PROGRAM SDOMotorErrorFlags
VAR
	ErrorFlagsKlemme1: getSDOMotorErrorFlags;
	ErrorFlagsKlemme2: getSDOMotorErrorFlags;
END_VAR

ErrorFlagsKlemme1.nSlaveAddr := 1002;
ErrorFlagsKlemme1();

END_PROGRAM

(* stored: Version 1.1.0.1, ProductVersion 3.1.4022.3
   POU SDOMotorErrorFlags: Id {009dd3da-fe0c-4125-961f-937488e6d44b}, SpecialFunc None *)
